// TIA Portal V20 export
FUNCTION_BLOCK "FB_MotorControl"   // FB1, SCL
{ S7_Optimized_Access := 'TRUE' }
VERSION : 0.2
// stored: MemoryReserve 100, SetENOAutomatically false
   VAR_INPUT
      bStart : Bool;
      bStop : Bool;
      bAutoStop : Bool;
   END_VAR
   VAR_OUTPUT
      bRunning : Bool;
      bFault : Bool;
   END_VAR
   VAR
      tRunTime : Time;
   END_VAR
BEGIN

   IF #bStart AND NOT #bStop AND NOT #bAutoStop THEN
       #bRunning := TRUE;
   END_IF;

   IF #bStop OR #bAutoStop THEN
       #bRunning := FALSE;
   END_IF;
END_FUNCTION_BLOCK
